// TIA Portal V17 export
// export: Created 2025-05-06T14:47:38.1340186Z, ExportSetting WithDefaults, DisplayName Totally Integrated Automation Portal, DisplayVersion V17 Update 8, DisplayName TIA Portal Openness, DisplayVersion V17 Update 8, DisplayName TIA Portal Version Control Interface, DisplayVersion V17, DisplayName SINAMICS Startdrive Advanced, DisplayVersion V17 SP2, DisplayName SINAMICS Startdrive G110M, G120, G120C, G120D, G120P, G115D, DisplayVersion V17 SP2, DisplayName SINAMICS Startdrive G130, G150, S120, S150, SINAMICS MV, S210, DisplayVersion V17 SP2, DisplayName STEP 7 Professional, DisplayVersion V17 Update 8, DisplayName SINUMERIK ONE STEP 7 Toolbox, DisplayVersion V17 Update 12, DisplayName SINUMERIK 840D sl STEP 7 Toolbox, DisplayVersion V17 Update 12, DisplayName STEP 7 Safety, DisplayVersion V17 Update 6, DisplayName WinCC Advanced, DisplayVersion V17 Update 8
FUNCTION_BLOCK "FB22108_POWDER_CURRENT_SENSOR"   // FB22108, LAD
{ S7_Optimized_Access := 'FALSE' }
VERSION : 0.1
// stored: AutoNumber false, IsIECCheckEnabled false, SetENOAutomatically false, UDAEnableTagReadback false
   VAR_INPUT
      SENSOR_VALUE : Int;   // SENSOR VALUE
      PF_LINE_ON : Bool;   // POWDER FEEDER LINE SWITCHED ON
   END_VAR
   VAR_OUTPUT
      CURRENT_LOW_LIMIT_ALARM : Bool;   // CURRENT LOW LIMIT ALARM
      CURRENT_HIGH_LIMIT_ALARM : Bool;   // CURRENT HIGH LIMIT ALARM
   END_VAR
   VAR DB_SPECIFIC
      OUTPUT : Struct
         POWDER_FILLING_STOP_BY_CURRENT : Bool;   // HMI POWDER FILLING STOP BY CURRENT
         POWDER_FILLING_START_BY_CURRENT : Bool;   // HMI POWDER FILLING START BY CURRENT
      END_STRUCT;
      INPUT_SETTINGS : Struct
         NORMALIZED_VALUE : Real;   // NORMALIZED
         SCALED_VALUE : Real;   // SCALED
      END_STRUCT;
      HMI : Struct
         HIGH_CURRENT_LIMIT : UInt;   // HMI HIGH CURRENT LIMIT
         LOW_CURRENT_LIMIT : UInt;   // HMI LOW CURRENT LIMIT
      END_STRUCT;
      INTERNAL : Struct
         CURRENT_AVG_BLCK_START : Real;   // CURRENT AVERAGE BLOCK START
         CURRENT_AVG_BLCK_STOP : Real;   // CURRENT AVERAGE BLOCK STOP
         ACTUAL_CURRENT_TO_START : Real;   // CURRENT AVERAGE BLOCK HMI START
         ACTUAL_CURRENT_TO_STOP : Real;   // CURRENT AVERAGE BLOCK HMI STOP
      END_STRUCT;
      ALARM_SETTINGS : Struct
         ALARM_LOW_LIMIT : Real;   // CURRENT BELOW LOW LIMT ALARM
         ALARM_HIGH_LIMIT : Real;   // CURRENT OVER HIGH LIMIT ALARM
      END_STRUCT;
   END_VAR
   VAR
      DB_CURRENT_AVERAGE_START : "FB22109_POWDER_CURRENT_AVG";
      DB_CURRENT_AVERAGE_STOP { S7_SetPoint := 'True'} : "FB22109_POWDER_CURRENT_AVG";
   END_VAR
   VAR DB_SPECIFIC
      START_BY_CURRENT_TIMER { S7_SetPoint := 'True'} : TON_TIME;
      CURRENT_HIGH_LIMIT_ALARM_TIMER { S7_SetPoint := 'True'} : TON_TIME;
      CURRENT_LOW_LIMIT_ALARM_TIMER { S7_SetPoint := 'True'} : TON_TIME;
   END_VAR
   // START_BY_CURRENT_TIMER.PT := T#1s;
   // CURRENT_HIGH_LIMIT_ALARM_TIMER.PT := T#1s;
   // CURRENT_LOW_LIMIT_ALARM_TIMER.PT := T#1s;
   VAR_TEMP   // added for the SCL form of the ladder/FBD networks
      _w1 : Bool;
   END_VAR
BEGIN

REGION Network 1: SCALE - CURRENT VALUE
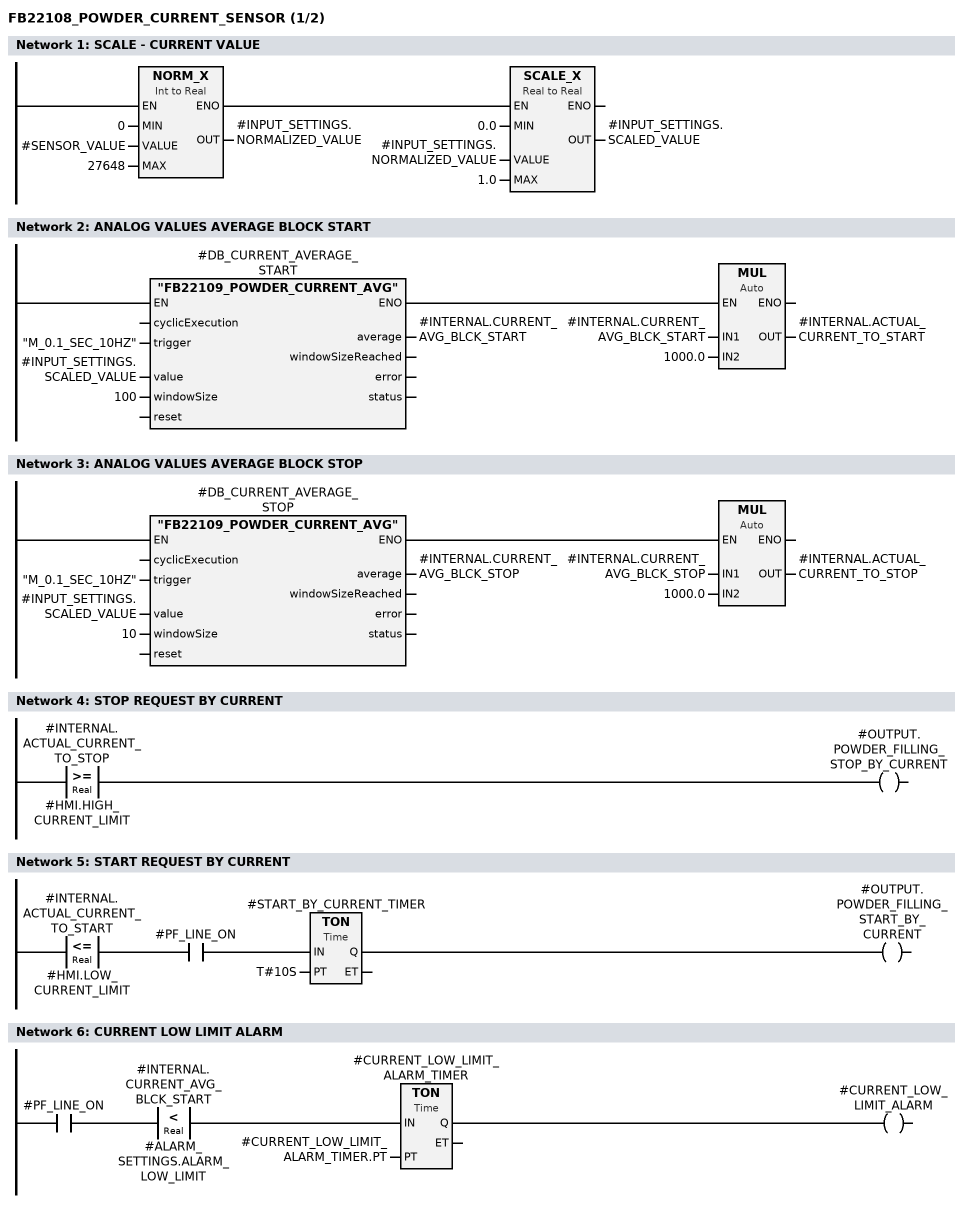
   RUNG wire#powerrail
      { S7_Templates := "[SrcType := Int, DestType := Real]"; S7_GenerateENO := "TRUE" } Normalize(min := 0, value := #SENSOR_VALUE, max := 27648, out => #INPUT_SETTINGS.NORMALIZED_VALUE)
      { S7_Templates := "[SrcType := Real, DestType := Real]"; S7_GenerateENO := "TRUE" } Scale(min := 0.0, value := #INPUT_SETTINGS.NORMALIZED_VALUE, max := 1.0, out => #INPUT_SETTINGS.SCALED_VALUE)
   END_RUNG
   // the same network as SCL:
   // ENO of a box is taken as its EN; it also drops when the box reports an error
   #INPUT_SETTINGS.NORMALIZED_VALUE := NORM_X(MIN := 0, VALUE := #SENSOR_VALUE, MAX := 27648);
   #INPUT_SETTINGS.SCALED_VALUE := SCALE_X(MIN := 0.0, VALUE := #INPUT_SETTINGS.NORMALIZED_VALUE, MAX := 1.0);
END_REGION

REGION Network 2: ANALOG VALUES AVERAGE BLOCK START
   RUNG wire#powerrail
      #DB_CURRENT_AVERAGE_START(cyclicExecution :=, trigger := "M_0.1_SEC_10HZ", value := #INPUT_SETTINGS.SCALED_VALUE, windowSize := 100, reset :=, average => #INTERNAL.CURRENT_AVG_BLCK_START, windowSizeReached =>, error =>, status =>)
      { S7_GenerateENO := "TRUE" } Mul(in1 := #INTERNAL.CURRENT_AVG_BLCK_START, in2 := 1000.0, out => #INTERNAL.ACTUAL_CURRENT_TO_START)
   END_RUNG
   // the same network as SCL:
   #DB_CURRENT_AVERAGE_START(trigger := "M_0.1_SEC_10HZ",   // "FB22109_POWDER_CURRENT_AVG"
                           value := #INPUT_SETTINGS.SCALED_VALUE,
                           windowSize := 100,
                           average => #INTERNAL.CURRENT_AVG_BLCK_START,
                           ENO => #_w1);
   IF #_w1 THEN #INTERNAL.ACTUAL_CURRENT_TO_START := #INTERNAL.CURRENT_AVG_BLCK_START * 1000.0; END_IF;
END_REGION

REGION Network 3: ANALOG VALUES AVERAGE BLOCK STOP
   RUNG wire#powerrail
      #DB_CURRENT_AVERAGE_STOP(cyclicExecution :=, trigger := "M_0.1_SEC_10HZ", value := #INPUT_SETTINGS.SCALED_VALUE, windowSize := 10, reset :=, average => #INTERNAL.CURRENT_AVG_BLCK_STOP, windowSizeReached =>, error =>, status =>)
      { S7_GenerateENO := "TRUE" } Mul(in1 := #INTERNAL.CURRENT_AVG_BLCK_STOP, in2 := 1000.0, out => #INTERNAL.ACTUAL_CURRENT_TO_STOP)
   END_RUNG
   // the same network as SCL:
   #DB_CURRENT_AVERAGE_STOP(trigger := "M_0.1_SEC_10HZ",   // "FB22109_POWDER_CURRENT_AVG"
                           value := #INPUT_SETTINGS.SCALED_VALUE,
                           windowSize := 10,
                           average => #INTERNAL.CURRENT_AVG_BLCK_STOP,
                           ENO => #_w1);
   IF #_w1 THEN #INTERNAL.ACTUAL_CURRENT_TO_STOP := #INTERNAL.CURRENT_AVG_BLCK_STOP * 1000.0; END_IF;
END_REGION

REGION Network 4: STOP REQUEST BY CURRENT
   RUNG wire#powerrail
      { S7_Templates := "SrcType := Real" } GE_Contact(in1 := #INTERNAL.ACTUAL_CURRENT_TO_STOP, in2 := #HMI.HIGH_CURRENT_LIMIT)
      Coil( #OUTPUT.POWDER_FILLING_STOP_BY_CURRENT )
   END_RUNG
   // the same network as SCL:
   #OUTPUT.POWDER_FILLING_STOP_BY_CURRENT := #INTERNAL.ACTUAL_CURRENT_TO_STOP >= #HMI.HIGH_CURRENT_LIMIT;
END_REGION

REGION Network 5: START REQUEST BY CURRENT
   RUNG wire#powerrail
      { S7_Templates := "SrcType := Real" } LE_Contact(in1 := #INTERNAL.ACTUAL_CURRENT_TO_START, in2 := #HMI.LOW_CURRENT_LIMIT)
      Contact( #PF_LINE_ON )
      { S7_Templates := "time_type := Time" } #START_BY_CURRENT_TIMER.TON(pt := T#10S, et =>)
      Coil( #OUTPUT.POWDER_FILLING_START_BY_CURRENT )
   END_RUNG
   // the same network as SCL:
   #START_BY_CURRENT_TIMER(IN := (#INTERNAL.ACTUAL_CURRENT_TO_START <= #HMI.LOW_CURRENT_LIMIT) AND #PF_LINE_ON,   // TON
                           PT := T#10S);
   #OUTPUT.POWDER_FILLING_START_BY_CURRENT := #START_BY_CURRENT_TIMER.Q;
END_REGION

REGION Network 6: CURRENT LOW LIMIT ALARM
   RUNG wire#powerrail
      Contact( #PF_LINE_ON )
      { S7_Templates := "SrcType := Real" } LT_Contact(in1 := #INTERNAL.CURRENT_AVG_BLCK_START, in2 := #ALARM_SETTINGS.ALARM_LOW_LIMIT)
      { S7_Templates := "time_type := Time" } #CURRENT_LOW_LIMIT_ALARM_TIMER.TON(pt := #CURRENT_LOW_LIMIT_ALARM_TIMER.PT, et =>)
      Coil( #CURRENT_LOW_LIMIT_ALARM )
   END_RUNG
   // the same network as SCL:
   #CURRENT_LOW_LIMIT_ALARM_TIMER(IN := #PF_LINE_ON AND (#INTERNAL.CURRENT_AVG_BLCK_START < #ALARM_SETTINGS.ALARM_LOW_LIMIT),   // TON
                           PT := #CURRENT_LOW_LIMIT_ALARM_TIMER.PT);
   #CURRENT_LOW_LIMIT_ALARM := #CURRENT_LOW_LIMIT_ALARM_TIMER.Q;
END_REGION

REGION Network 7: CURRENT HIGH LIMIT ALARM
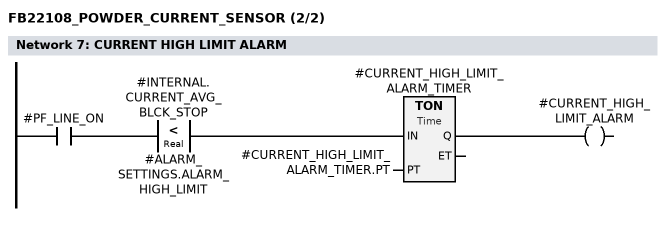
   RUNG wire#powerrail
      Contact( #PF_LINE_ON )
      { S7_Templates := "SrcType := Real" } LT_Contact(in1 := #INTERNAL.CURRENT_AVG_BLCK_STOP, in2 := #ALARM_SETTINGS.ALARM_HIGH_LIMIT)
      { S7_Templates := "time_type := Time" } #CURRENT_HIGH_LIMIT_ALARM_TIMER.TON(pt := #CURRENT_HIGH_LIMIT_ALARM_TIMER.PT, et =>)
      Coil( #CURRENT_HIGH_LIMIT_ALARM )
   END_RUNG
   // the same network as SCL:
   #CURRENT_HIGH_LIMIT_ALARM_TIMER(IN := #PF_LINE_ON AND (#INTERNAL.CURRENT_AVG_BLCK_STOP < #ALARM_SETTINGS.ALARM_HIGH_LIMIT),   // TON
                           PT := #CURRENT_HIGH_LIMIT_ALARM_TIMER.PT);
   #CURRENT_HIGH_LIMIT_ALARM := #CURRENT_HIGH_LIMIT_ALARM_TIMER.Q;
END_REGION
END_FUNCTION_BLOCK
